// TwinCAT 3 PLC project TcAbbLinkinPLC
// Title: TcAbbLinkin
// Company: Loupe
// Author: Loupe
// ProjectVersion: 0.1.0
// ProgramVersion: 3.1.4024.0
// libraries:
//   Tc2_Standard, * (Beckhoff Automation GmbH)
//   Tc2_System, * (Beckhoff Automation GmbH)
//   Tc2_Utilities, * (Beckhoff Automation GmbH)
//   Tc3_IotBase, * (Beckhoff Automation GmbH)
//   Tc3_JsonXml, * (Beckhoff Automation GmbH)
//   Tc3_Module, * (Beckhoff Automation GmbH)
// project tree:
//   DUTs/ AbbLinkinAuthDigest_Typ.TcDUT, AbbLinkinConfiguration_Typ.TcDUT, AbbLinkinRequestResults_Typ.TcDUT, AbbLinkinRequest_Typ.TcDUT, AbbLinkinRequestQueue_Typ.TcDUT, AbbLinkinRequestStatus_Typ.TcDUT, AbbLinkinAuth_Typ.TcDUT, ABBLINKIN_AUTH_HEADER_VALUE.TcDUT, ABBLINKIN_RWS_API_VERSION.TcDUT, ABBLINKIN_STATE.TcDUT, ABBLINKIN_COMMAND_TYPE.TcDUT, ABBLINKIN_DATA_TYPE_Typ.TcDUT, ABBLINKIN_STRING_EX_LEN.TcDUT (not stored)
//   / PlcTask.TcTTO
//   POUs/ MAIN.TcPOU, Example.TcPOU, TcAbbLinkin.TcPOU
// real-time tasks:
//   TASK PlcTask: cycle T#10ms, priority 20, ADS port 350

CONFIGURATION TcAbbLinkinPLC
    RESOURCE PLC ON TwinCAT3
        TASK PlcTask(INTERVAL := T#10ms, PRIORITY := 20);
        PROGRAM MAIN WITH PlcTask : MAIN;
    END_RESOURCE
END_CONFIGURATION

// ---- DUTs/AbbLinkinAuthDigest_Typ.TcDUT
// Copyright (c) 2024 Loupe (https://loupe.team), provided under the MIT License.
TYPE AbbLinkinAuthDigest_Typ :
STRUCT
	realm : STRING;
	qop : STRING;
	nonce : STRING;
	opaque : STRING;
	nc : STRING;
	cnonce : STRING;
	response : STRING;
	authContent : ABBLINKIN_STRING_EX_LEN;
END_STRUCT
END_TYPE

// ---- DUTs/AbbLinkinConfiguration_Typ.TcDUT
// Copyright (c) 2024 Loupe (https://loupe.team), provided under the MIT License.
TYPE AbbLinkinConfiguration_Typ :
STRUCT
	rwsIpAddress : STRING := '127.0.0.1';
	rwsTcpPort : USINT := 80;
	rwsVersion : ABBLINKIN_RWS_API_VERSION;
	rwsUsername : STRING := 'Default User';
	rwsPassword : STRING := 'robotics';
	tlsAllowRwsCertSelfSigned : BOOL := FALSE;
	tlsCAFile : STRING := '';
END_STRUCT
END_TYPE

// ---- DUTs/AbbLinkinRequestResults_Typ.TcDUT
// Copyright (c) 2024 Loupe (https://loupe.team), provided under the MIT License.
TYPE AbbLinkinRequestResults_Typ :
STRUCT
	pDataBool	: POINTER TO BOOL;
	pDataDint	: POINTER TO DINT;
	pDataLreal	: POINTER TO LREAL;
	pDataString	: POINTER TO STRING;
	dataType	: ABBLINKIN_DATA_TYPE_Typ;
	dataLen		: INT;
END_STRUCT
END_TYPE

// ---- DUTs/AbbLinkinRequest_Typ.TcDUT
// Copyright (c) 2024 Loupe (https://loupe.team), provided under the MIT License.
TYPE AbbLinkinRequest_Typ :
STRUCT
	command : ABBLINKIN_COMMAND_TYPE;
	uri : STRING;
	httpMethod : ETcIotHttpRequestType;
	httpBody : ABBLINKIN_STRING_EX_LEN := '';
	pStatus : POINTER TO AbbLinkinRequestStatus_Typ;
	results : AbbLinkinRequestResults_Typ;
END_STRUCT
END_TYPE

// ---- DUTs/AbbLinkinRequestQueue_Typ.TcDUT
// Copyright (c) 2024 Loupe (https://loupe.team), provided under the MIT License.
TYPE AbbLinkinRequestQueue_Typ :
STRUCT
	request : AbbLinkinRequest_Typ;
	empty : BOOL := TRUE;
END_STRUCT
END_TYPE

// ---- DUTs/AbbLinkinRequestStatus_Typ.TcDUT
// Copyright (c) 2024 Loupe (https://loupe.team), provided under the MIT License.
TYPE AbbLinkinRequestStatus_Typ :
STRUCT
	busy		: BOOL;
	done		: BOOL;
	error		: BOOL;
	errorID		: DINT;
	errorMsg	: STRING;
END_STRUCT
END_TYPE

// ---- DUTs/AbbLinkinAuth_Typ.TcDUT
// Copyright (c) 2024 Loupe (https://loupe.team), provided under the MIT License.
TYPE AbbLinkinAuth_Typ :
STRUCT
	numAttempts : UINT;
	wwwAuthContent : ABBLINKIN_STRING_EX_LEN;
	digest : AbbLinkinAuthDigest_Typ;
	httpSessionCookie : STRING;
	ABBCXCookie : STRING;
END_STRUCT
END_TYPE

// ---- DUTs/ABBLINKIN_AUTH_HEADER_VALUE.TcDUT
{attribute 'qualified_only'}
{attribute 'strict'}
TYPE ABBLINKIN_AUTH_HEADER_VALUE :
(
	NONE,
	BASIC,
	DIGEST
);
END_TYPE

// ---- DUTs/ABBLINKIN_RWS_API_VERSION.TcDUT
{attribute 'qualified_only'}
{attribute 'strict'}
TYPE ABBLINKIN_RWS_API_VERSION :
(
	V1 := 0,
	V2 := 2
);
END_TYPE

// ---- DUTs/ABBLINKIN_STATE.TcDUT
// Copyright (c) 2024 Loupe (https://loupe.team), provided under the MIT License.
{attribute 'qualified_only'}
{attribute 'strict'}
TYPE ABBLINKIN_STATE :
(
	IDLE,
	SEND_REQUEST,
	WAIT_FOR_RESONSE,
	PROCESS_RESPONSE,
	AUTH_START,
	AUTH_SEND_REQUEST,
	AUTH_WAIT_FOR_RESONSE,
	AUTH_PROCESS_RESPONSE,
	AUTH_DIGEST_RESPONSE_CALCULATE,
	AUTH_DIGEST_RESPONSE_SEND
);
END_TYPE

// ---- DUTs/ABBLINKIN_COMMAND_TYPE.TcDUT
// Copyright (c) 2024 Loupe (https://loupe.team), provided under the MIT License.
{attribute 'qualified_only'}
{attribute 'strict'}
TYPE ABBLINKIN_COMMAND_TYPE :
(
	GET_IO,
	GET_PANEL_CTRL_STATE,
	GET_PANEL_OP_MODE,
	GET_RAPID_STATE,
	GET_SYMBOL,
	POWER_OFF,
	POWER_ON,
	RAPID_RESET,
	RAPID_START,
	RAPID_STOP,
	SET_IO,
	SET_SYMBOL
);
END_TYPE

// ---- DUTs/ABBLINKIN_DATA_TYPE_Typ.TcDUT
// Copyright (c) 2024 Loupe (https://loupe.team), provided under the MIT License.
{attribute 'qualified_only'}
{attribute 'strict'}
TYPE ABBLINKIN_DATA_TYPE_Typ :
(
	_NONE,
	_STRING,
	_BOOL,
	_DINT,
	_LREAL
);
END_TYPE

// ---- POUs/MAIN.TcPOU
// Copyright (c) 2024 Loupe (https://loupe.team), provided under the MIT License.
PROGRAM MAIN
VAR
	myRobotLink : TcAbbLinkin;
	userSetConfigurationNow : BOOL := TRUE;
	userConnectStartNow : BOOL := TRUE;
	userConnectStopNow : BOOL;
	
	userGetPanelCtrlStateNow : BOOL;
	userGetPanelCtrlStateStatus : AbbLinkinRequestStatus_Typ;
	userGetPanelCtrlStateResult : STRING;
	
	userGetPanelOpModeNow : BOOL;
	userGetPanelOpModeStatus : AbbLinkinRequestStatus_Typ;
	userGetPanelOpModeResult : STRING;
	
	userGetRapidStateNow : BOOL;
	userGetRapidStateStatus : AbbLinkinRequestStatus_Typ;
	userGetRapidStateResult : STRING;
	
	userGetIoBoolNow : BOOL;
	userGetIoBoolStatus : AbbLinkinRequestStatus_Typ;
	userGetIoBoolResult : BOOL;
	
	userGetIoLrealNow : BOOL;
	userGetIoLrealStatus : AbbLinkinRequestStatus_Typ;
	userGetIoLrealResult : LREAL;
	
	userGetIoDintNow : BOOL;
	userGetIoDintStatus : AbbLinkinRequestStatus_Typ;
	userGetIoDintResult : DINT;
	
	
	userSetIoBoolNow : BOOL;
	userSetIoBoolValue : BOOL := 1;
	userSetIoBoolStatus : AbbLinkinRequestStatus_Typ;
	userSetIoDintNow : BOOL;
	userSetIoDintValue : DINT := 57;
	userSetIoDintStatus : AbbLinkinRequestStatus_Typ;
	userSetIoLrealNow : BOOL;
	userSetIoLrealValue : LREAL := 41.123456;
	userSetIoLrealStatus : AbbLinkinRequestStatus_Typ;
	
	
	userGetSymbolBoolNow : BOOL;
	userGetSymbolBoolResult : BOOL;
	userGetSymbolBoolStatus : AbbLinkinRequestStatus_Typ;
	userGetSymbolNumNow : BOOL;
	userGetSymbolNumResult : LREAL;
	userGetSymbolNumStatus : AbbLinkinRequestStatus_Typ;
	userGetSymbolStringNow : BOOL;
	userGetSymbolStringResult : STRING;
	userGetSymbolStringStatus : AbbLinkinRequestStatus_Typ;
	
	userSetSymbolBoolNow : BOOL;
	userSetSymbolBoolValue : BOOL := 1;
	userSetSymbolBoolStatus : AbbLinkinRequestStatus_Typ;
	userSetSymbolDintNow : BOOL;
	userSetSymbolDintValue : DINT := -57;
	userSetSymbolDintStatus : AbbLinkinRequestStatus_Typ;
	userSetSymbolLrealNow : BOOL;
	userSetSymbolLrealValue : LREAL := -41.123456;
	userSetSymbolLrealStatus : AbbLinkinRequestStatus_Typ;
	userSetSymbolStringNow : BOOL;
	userSetSymbolStringValue : STRING := 'test String';
	userSetSymbolStringStatus : AbbLinkinRequestStatus_Typ;
	userSetSymbolWStringNow : BOOL;
	userSetSymbolWStringValue : WSTRING := "test WString";
	userSetSymbolWStringStatus : AbbLinkinRequestStatus_Typ;
	
	
	userPowerOffNow : BOOL;
	userPowerOffStatus : AbbLinkinRequestStatus_Typ;
	userPowerOnNow : BOOL;
	userPowerOnStatus : AbbLinkinRequestStatus_Typ;
	userRapidResetNow : BOOL;
	userRapidResetStatus : AbbLinkinRequestStatus_Typ;
	userRapidStopNow : BOOL;
	userRapidStopStatus : AbbLinkinRequestStatus_Typ;
	userRapidStartNow : BOOL;
	userRapidStartStatus : AbbLinkinRequestStatus_Typ;
	
	
	userAckErrorNow : BOOL;
END_VAR


// Set configuration
if userSetConfigurationNow then
	myRobotLink.configuration.rwsIpAddress := '127.0.0.1';
	myRobotLink.configuration.rwsTcpPort := 80;
	myRobotLink.configuration.rwsVersion := ABBLINKIN_RWS_API_VERSION.V2;
	myRobotLink.configuration.rwsUsername := 'Default User';
	myRobotLink.configuration.rwsPassword := 'robotics';
	//myRobotLink.configuration.tlsAllowRwsCertSelfSigned := TRUE;
	myRobotLink.configuration.tlsAllowRwsCertSelfSigned := FALSE;
	myRobotLink.configuration.tlsCAFile := 'C:\TwinCAT\3.1\Config\Certificates\TcAbbLinkinCA.pem';
	
	userSetConfigurationNow := FALSE;
END_IF


// Cyclic
myRobotLink.Cyclic();


IF userConnectStartNow THEN
	myRobotLink.Connect();
	userConnectStartNow := FALSE;
END_IF

IF userConnectStopNow THEN
	myRobotLink.Disconnect();
	userConnectStopNow := FALSE;
END_IF


IF userGetPanelCtrlStateNow THEN
	myRobotLink.GetPanelCtrlState(ADR(userGetPanelCtrlStateStatus), ADR(userGetPanelCtrlStateResult));
	userGetPanelCtrlStateNow := FALSE;
END_IF


IF userGetPanelOpModeNow THEN
	myRobotLink.GetPanelOpMode(ADR(userGetPanelOpModeStatus), ADR(userGetPanelOpModeResult));
	userGetPanelOpModeNow := FALSE;
END_IF


IF userGetRapidStateNow THEN
	myRobotLink.GetRapidState(ADR(userGetRapidStateStatus), ADR(userGetRapidStateResult));
	userGetRapidStateNow := FALSE;
END_IF


IF userGetIoBoolNow THEN
	myRobotLink.GetIODigital(signal := 'myInputDIG', pStatus := ADR(userGetIoBoolStatus), pResult := ADR(userGetIoBoolResult));
	userGetIoBoolNow := FALSE;
END_IF

IF userGetIoLrealNow THEN
	myRobotLink.GetIOAnalog(signal := 'myInputANA', pStatus := ADR(userGetIoLrealStatus), pResult := ADR(userGetIoLrealResult));
	userGetIoLrealNow := FALSE;
END_IF

IF userGetIoDintNow THEN
	myRobotLink.GetIOGroup(signal := 'myInputGRP', pStatus := ADR(userGetIoDintStatus), pResult := ADR(userGetIoDintResult));
	userGetIoDintNow := FALSE;
END_IF


IF userSetIoBoolNow THEN
	myRobotLink.SetIO('myInputDIG', userSetIoBoolValue, ADR(userSetIoBoolStatus));
	userSetIoBoolNow := FALSE;
END_IF
IF userSetIoDintNow THEN
	myRobotLink.SetIO('myInputGRP', userSetIoDintValue, ADR(userSetIoDintStatus));
	userSetIoDintNow := FALSE;
END_IF
IF userSetIoLrealNow THEN
	myRobotLink.SetIO('myInputANA', userSetIoLrealValue, ADR(userSetIoLrealStatus));
	userSetIoLrealNow := FALSE;
END_IF


IF userGetSymbolBoolNow THEN
	myRobotLink.GetSymbolBool(symbolUrl := 'RAPID/T_ROB1/Module1/myRapidBool', pStatus := ADR(userGetSymbolBoolStatus), pResult := ADR(userGetSymbolBoolResult));
	userGetSymbolBoolNow := FALSE;
END_IF
IF userGetSymbolNumNow THEN
	myRobotLink.GetSymbolNum(symbolUrl := 'RAPID/T_ROB1/Module1/myRapidNum', pStatus := ADR(userGetSymbolNumStatus), pResult := ADR(userGetSymbolNumResult));
	userGetSymbolNumNow := FALSE;
END_IF
IF userGetSymbolStringNow THEN
	myRobotLink.GetSymbolString(symbolUrl := 'RAPID/T_ROB1/Module1/myRapidString', pStatus := ADR(userGetSymbolStringStatus), pResult := ADR(userGetSymbolStringResult));
	userGetSymbolStringNow := FALSE;
END_IF


IF userSetSymbolBoolNow THEN
	myRobotLink.SetSymbol('RAPID/T_ROB1/Module1/myRapidBool', userSetSymbolBoolValue, ADR(userSetSymbolBoolStatus));
	userSetSymbolBoolNow := FALSE;
END_IF
IF userSetSymbolDintNow THEN
	myRobotLink.SetSymbol('RAPID/T_ROB1/Module1/myRapidNum', userSetSymbolDintValue, ADR(userSetSymbolDintStatus));
	userSetSymbolDintNow := FALSE;
END_IF
IF userSetSymbolLrealNow THEN
	myRobotLink.SetSymbol('RAPID/T_ROB1/Module1/myRapidNum', userSetSymbolLrealValue, ADR(userSetSymbolLrealStatus));
	userSetSymbolLrealNow := FALSE;
END_IF
IF userSetSymbolStringNow THEN
	myRobotLink.SetSymbol('RAPID/T_ROB1/Module1/myRapidString', userSetSymbolStringValue, ADR(userSetSymbolStringStatus));
	userSetSymbolStringNow := FALSE;
END_IF
IF userSetSymbolWStringNow THEN
	myRobotLink.SetSymbol('RAPID/T_ROB1/Module1/myRapidString', userSetSymbolWStringValue, ADR(userSetSymbolWStringStatus));
	userSetSymbolWStringNow := FALSE;
END_IF


IF userPowerOffNow THEN
	myRobotLink.PowerOff(ADR(userPowerOffStatus));
	userPowerOffNow := FALSE;
END_IF
IF userPowerOnNow THEN
	myRobotLink.PowerOn(ADR(userPowerOnStatus));
	userPowerOnNow := FALSE;
END_IF
IF userRapidResetNow THEN
	myRobotLink.RapidReset(ADR(userRapidResetStatus));
	userRapidResetNow := FALSE;
END_IF
IF userRapidStopNow THEN
	myRobotLink.RapidStop(ADR(userRapidStopStatus));
	userRapidStopNow := FALSE;
END_IF
IF userRapidStartNow THEN
	myRobotLink.RapidStart(ADR(userRapidStartStatus));
	userRapidStartNow := FALSE;
END_IF


IF userAckErrorNow THEN
	myRobotLink.AckError();
	userAckErrorNow := FALSE;
END_IF

END_PROGRAM

// ---- POUs/TcAbbLinkin.TcPOU
// Copyright (c) 2024 Loupe (https://loupe.team), provided under the MIT License.
FUNCTION_BLOCK TcAbbLinkin
VAR_INPUT
	configuration : AbbLinkinConfiguration_Typ;
END_VAR
VAR_OUTPUT
	readyForCmd : BOOL;
	error : BOOL;
	errorID : DINT;
	errorMsg : STRING;
END_VAR
VAR
	_connectionEnable : BOOL;
	_sendingEnabled : BOOL;
	_authorized : BOOL;
	
	_httpClient : FB_IotHttpClient;
	_httpRequest : FB_IotHttpRequest;
	_httpHeader : FB_IotHttpHeaderFieldMap;
	
	_methodConnectionStartCalled : BOOL;
	_methodConnectionStopCalled : BOOL;
	_methodAckErrorCalled : BOOL;
	
	_state : ABBLINKIN_STATE;
	_auth : AbbLinkinAuth_Typ;
	_requestQueue : AbbLinkinRequestQueue_Typ;
	_currentRequest : AbbLinkinRequest_Typ;
	_numRequestAttempts : UINT;
END_VAR

VAR CONSTANT
	AUTH_URI : STRING := '/?json=1';
	MAX_REQUESTS_ATTEMPTS : UINT := 3;
END_VAR

// Copyright (c) 2024 Loupe (https://loupe.team), provided under the MIT License.
METHOD PRIVATE _calculateDigestResponse : STRING
VAR_INPUT
	username : STRING;
	realm : STRING;
	password : STRING;
	httpMethod : STRING;
	uri : STRING;
	nonce : STRING;
	nc : STRING;
	cnonce : STRING;
	qop : STRING;
END_VAR

VAR
	tempString : ABBLINKIN_STRING_EX_LEN;
	h1_byArr : ARRAY[0..15] OF BYTE;
	h1_hexStr : STRING;
	h2_byArr : ARRAY[0..15] OF BYTE;
	h2_hexStr : STRING;
	response_byArr : ARRAY[0..15] OF BYTE;
	response_hexStr : STRING;
	i : INT;
END_VAR

// H1 hash
tempString := '';
tempString := CONCAT(tempString, username);
tempString := CONCAT(tempString, ':');
tempString := CONCAT(tempString, realm);
tempString := CONCAT(tempString, ':');
tempString := CONCAT(tempString, password);
F_GenerateHashValue(E_HashMode.HASH_MD5, ADR(tempString), INT_TO_UDINT(LEN(tempString)), ADR(h1_byArr), SIZEOF(h1_byArr));
h1_hexStr := '';
FOR i := 0 TO 15 DO
	h1_hexStr := CONCAT(h1_hexStr, BYTE_TO_HEXSTR(h1_byArr[i], 2, TRUE));
END_FOR


// H2 Hash
tempString := '';
tempString := CONCAT(tempString, httpMethod);
tempString := CONCAT(tempString, ':');
tempString := CONCAT(tempString, uri);
F_GenerateHashValue(E_HashMode.HASH_MD5, ADR(tempString), INT_TO_UDINT(LEN(tempString)), ADR(h2_byArr), SIZEOF(h2_byArr));
h2_hexStr := '';
FOR i := 0 TO 15 DO
	h2_hexStr := CONCAT(h2_hexStr, BYTE_TO_HEXSTR(h2_byArr[i], 2, TRUE));
END_FOR


// Response hash
tempString := '';
tempString := CONCAT(tempString, h1_hexStr);
tempString := CONCAT(tempString, ':');
tempString := CONCAT(tempString, nonce);
tempString := CONCAT(tempString, ':');
tempString := CONCAT(tempString, nc);
tempString := CONCAT(tempString, ':');
tempString := CONCAT(tempString, cnonce);
tempString := CONCAT(tempString, ':');
tempString := CONCAT(tempString, qop);
tempString := CONCAT(tempString, ':');
tempString := CONCAT(tempString, h2_hexStr);
F_GenerateHashValue(E_HashMode.HASH_MD5, ADR(tempString), INT_TO_UDINT(LEN(tempString)), ADR(response_byArr), SIZEOF(response_byArr));
response_hexStr := '';
FOR i := 0 TO 15 DO
	response_hexStr := CONCAT(response_hexStr, BYTE_TO_HEXSTR(response_byArr[i], 2, TRUE));
END_FOR

_calculateDigestResponse := response_hexStr;
END_METHOD

// Copyright (c) 2024 Loupe (https://loupe.team), provided under the MIT License.
METHOD PRIVATE _callCommandSuccessHandler : BOOL
VAR_IN_OUT
	request : AbbLinkinRequest_Typ;
	httpRequest : FB_IotHttpRequest;
END_VAR

CASE request.command OF 
	ABBLINKIN_COMMAND_TYPE.GET_IO:
		_getIORespCallbackSuccess(httpRequest, request);
		
	ABBLINKIN_COMMAND_TYPE.GET_CTRL_STATE:
		_getCtrlStateRespCallbackSuccess(httpRequest, request);
		
	ABBLINKIN_COMMAND_TYPE.GET_OP_MODE:
		_getOpModeRespCallbackSuccess(httpRequest, request);
		
	ABBLINKIN_COMMAND_TYPE.GET_RAPID_STATE:
		_getRapidStateRespCallbackSuccess(httpRequest, request);
		
	ABBLINKIN_COMMAND_TYPE.GET_SYMBOL:
		_getSymbolRespCallbackSuccess(httpRequest, request);
		
	ABBLINKIN_COMMAND_TYPE.POWER_OFF:
		;// Do Nothing
		
	ABBLINKIN_COMMAND_TYPE.POWER_ON:
		;// Do Nothing
		
	ABBLINKIN_COMMAND_TYPE.RAPID_RESET:
		;// Do Nothing
		
	ABBLINKIN_COMMAND_TYPE.RAPID_START:
		;// Do Nothing
		
	ABBLINKIN_COMMAND_TYPE.RAPID_STOP:
		;// Do Nothing
		
	ABBLINKIN_COMMAND_TYPE.SET_IO:
		;// Do Nothing
		
	ABBLINKIN_COMMAND_TYPE.SET_SYMBOL:
		;// Do Nothing
		
END_CASE
END_METHOD

// Copyright (c) 2024 Loupe (https://loupe.team), provided under the MIT License.
METHOD PRIVATE _clearRequestStatus : BOOL
VAR_INPUT
	pStatus : POINTER TO AbbLinkinRequestStatus_Typ;
END_VAR

pStatus^.busy := FALSE;
pStatus^.done := FALSE;
pStatus^.error := FALSE;
pStatus^.errorID := 0;
pStatus^.errorMsg := '';

_clearRequestStatus := TRUE;
END_METHOD

// Copyright (c) 2024 Loupe (https://loupe.team), provided under the MIT License.
METHOD PRIVATE _configureClient : BOOL
VAR_IN_OUT
	connectionConfig : AbbLinkinConfiguration_Typ;	
END_VAR

_httpClient.sHostName := connectionConfig.rwsIpAddress;
_httpClient.nHostPort := connectionConfig.rwsTcpPort;
_httpClient.bKeepAlive := TRUE;
_httpClient.tConnectionTimeout := T#10S;


CASE connectionConfig.rwsVersion OF
	ABBLINKIN_RWS_API_VERSION.V1:
		_httpClient.stTLS.bNoServerCertCheck := FALSE;
		
	ABBLINKIN_RWS_API_VERSION.V2:
		IF connectionConfig.tlsAllowRwsCertSelfSigned THEN 
			_httpClient.stTLS.bNoServerCertCheck := TRUE;
		ELSE
			_httpClient.stTLS.bNoServerCertCheck := FALSE;
			_httpClient.stTLS.sCA := connectionConfig.tlsCAFile;
		END_IF
END_CASE
END_METHOD

// Copyright (c) 2024 Loupe (https://loupe.team), provided under the MIT License.
METHOD PRIVATE _encodeBase64 : STRING
VAR_INPUT
	rawText : STRING;
END_VAR
VAR
	_jsonDomParser : FB_JsonDomParser;
	_jsonRoot : SJsonValue;
	_jsonValue : SJsonValue;
	_jsonValue2 : SJsonValue;
END_VAR
	
_jsonRoot := _jsonDomParser.ParseDocument('{"k": ""}');
_jsonValue := _jsonDomParser.FindMember(_jsonRoot, 'k');
_jsonValue2 := _jsonDomParser.SetBase64(_jsonValue, ADR(rawText), LEN(rawText));
_encodeBase64 := _jsonDomParser.GetString(_jsonValue2);
END_METHOD

METHOD PRIVATE _generateCnonce : STRING
VAR_INPUT
END_VAR

_generateCnonce := 'diddLOPR';	// TODO: reimplement with random generation
END_METHOD

// Copyright (c) 2024 Loupe (https://loupe.team), provided under the MIT License.
METHOD PRIVATE _getCtrlStateRespCallbackSuccess : BOOL
VAR_IN_OUT
	httpRequest : FB_IotHttpRequest;
	request : AbbLinkinRequest_Typ;
END_VAR
VAR
	jsonDomParser : FB_JsonDomParser;
	jsonRoot : SJsonValue;
	jsonValue : SJsonValue;
	valuePath : STRING;
	tempString : STRING;
END_VAR
CASE configuration.rwsVersion OF 
	ABBLINKIN_RWS_API_VERSION.V1:
		valuePath := '_embedded/_state#0/ctrlstate';
	ABBLINKIN_RWS_API_VERSION.V2:
		valuePath := 'state#0/ctrlstate';
END_CASE

jsonRoot := httpRequest.GetJsonDomContent(jsonDomParser);
jsonValue := jsonDomParser.FindMemberPath(jsonRoot, valuePath);
IF (jsonValue <> 0) THEN
	request.results.pDataString^ := jsonDomParser.GetString(jsonValue);
ELSE
	request.pStatus^.error := TRUE;
	request.pStatus^.errorID := 0;
	request.pStatus^.errorMsg := 'Unable to parse RWS json response';
END_IF


_getCtrlStateRespCallbackSuccess := TRUE;
END_METHOD

// Copyright (c) 2024 Loupe (https://loupe.team), provided under the MIT License.
METHOD PRIVATE _getIO : BOOL
VAR_INPUT
	signal : STRING;
	pStatus : POINTER TO AbbLinkinRequestStatus_Typ;
	pResultBool : POINTER TO BOOL := 0;
	pResultDint : POINTER TO DINT := 0;
	pResultLreal : POINTER TO LREAL := 0;
END_VAR

VAR
	request : AbbLinkinRequest_Typ;
	pointersSet : INT;
END_VAR

VAR CONSTANT
	THIS_COMMAND_TYPE: ABBLINKIN_COMMAND_TYPE := ABBLINKIN_COMMAND_TYPE.GET_IO;
END_VAR
IF pStatus = 0 THEN
	_getIO := FALSE;
	RETURN;
END_IF

// Clear Status
_clearRequestStatus(pStatus);

// Check that one and only one pointer is populated
pointersSet := 0;
IF (pResultBOOL <> 0) THEN 
	request.results.dataType := ABBLINKIN_DATA_TYPE_Typ._BOOL;
	request.results.pDataBool := pResultBool;
	pointersSet := pointersSet + 1; 
END_IF
IF (pResultDINT <> 0) THEN
	request.results.dataType := ABBLINKIN_DATA_TYPE_Typ._DINT;
	request.results.pDataDint := pResultDint;
	pointersSet := pointersSet + 1;
END_IF
IF (pResultLREAL <> 0) THEN
	request.results.dataType := ABBLINKIN_DATA_TYPE_Typ._LREAL;
	request.results.pDataLreal := pResultLreal;
	pointersSet := pointersSet + 1;
END_IF


IF pointersSet = 0 THEN
	pStatus^.error := TRUE;
	pStatus^.errorMsg := TO_STRING(THIS_COMMAND_TYPE);
	pStatus^.errorMsg := CONCAT(pStatus^.errorMsg, ' : No result pointer set');
	_getIO := FALSE;
ELSIF pointersSet >= 2 THEN
	pStatus^.error := TRUE;
	pStatus^.errorMsg := TO_STRING(THIS_COMMAND_TYPE);
	pStatus^.errorMsg := CONCAT(pStatus^.errorMsg, ' : Two or more result pointer set');
	_getIO := FALSE;
END_IF

request.pStatus := pStatus;
request.command := THIS_COMMAND_TYPE;
request.httpMethod :=  ETcIotHttpRequestType.HTTP_Get;

CASE configuration.rwsVersion OF
	ABBLINKIN_RWS_API_VERSION.V1:
		request.uri := '/rw/iosystem/signals/';
		request.uri := CONCAT(request.uri, signal);
		request.uri := CONCAT(request.uri, '?json=1');

	ABBLINKIN_RWS_API_VERSION.V2:	
		request.uri := '/rw/iosystem/signals/';
		request.uri := CONCAT(request.uri, signal);
END_CASE

// Add Request to Queue, and Set Busy (or Error) Status
IF _requestQueueAdd(request) THEN
	pStatus^.busy := TRUE;
	_getIO := TRUE;
ELSE
	pStatus^.error := TRUE;
	pStatus^.errorMsg := TO_STRING(THIS_COMMAND_TYPE);
	pStatus^.errorMsg := CONCAT(pStatus^.errorMsg, ' could not be added to request Queue');
	_getIO := FALSE;
END_IF
END_METHOD

// Copyright (c) 2024 Loupe (https://loupe.team), provided under the MIT License.
METHOD PRIVATE _getIORespCallbackSuccess : BOOL
VAR_IN_OUT
	httpRequest : FB_IotHttpRequest;
	request : AbbLinkinRequest_Typ;
END_VAR
VAR
	jsonDomParser : FB_JsonDomParser;
	jsonRoot : SJsonValue;
	jsonValue : SJsonValue;
	valuePath : STRING;
	valueString : STRING;
END_VAR

CASE configuration.rwsVersion OF 
	ABBLINKIN_RWS_API_VERSION.V1:
		valuePath := '_embedded/_state#0/lvalue';
	ABBLINKIN_RWS_API_VERSION.V2:
		valuePath := '_embedded/resources#0/lvalue';
END_CASE

jsonRoot := httpRequest.GetJsonDomContent(jsonDomParser);
jsonValue := jsonDomParser.FindMemberPath(jsonRoot, valuePath);
IF (jsonValue <> 0) THEN
	valueString := jsonDomParser.GetString(jsonValue);
	
	CASE request.results.dataType OF
		ABBLINKIN_DATA_TYPE_Typ._BOOL:
			request.results.pDataBool^ := INT_TO_BOOL(STRING_TO_INT(valueString));
		ABBLINKIN_DATA_TYPE_Typ._DINT:
			request.results.pDataDint^ := STRING_TO_DINT(valueString);
		ABBLINKIN_DATA_TYPE_Typ._LREAL:
			request.results.pDataLreal^ := STRING_TO_LREAL(valueString);
	END_CASE
ELSE
	request.pStatus^.error := TRUE;
	request.pStatus^.errorID := 0;
	request.pStatus^.errorMsg := 'Unable to parse RWS json response';
END_IF


_getIORespCallbackSuccess := TRUE;
END_METHOD

// Copyright (c) 2024 Loupe (https://loupe.team), provided under the MIT License.
METHOD PRIVATE _getOpModeRespCallbackSuccess : BOOL
VAR_IN_OUT
	httpRequest : FB_IotHttpRequest;
	request : AbbLinkinRequest_Typ;
END_VAR
VAR
	jsonDomParser : FB_JsonDomParser;
	jsonRoot : SJsonValue;
	jsonValue : SJsonValue;
	valuePath : STRING;
	tempString : STRING;
END_VAR
CASE configuration.rwsVersion OF 
	ABBLINKIN_RWS_API_VERSION.V1:
		valuePath := '_embedded/_state#0/opmode';
	ABBLINKIN_RWS_API_VERSION.V2:
		valuePath := 'state#0/opmode';
END_CASE

jsonRoot := httpRequest.GetJsonDomContent(jsonDomParser);
jsonValue := jsonDomParser.FindMemberPath(jsonRoot, valuePath);
IF (jsonValue <> 0) THEN
	request.results.pDataString^ := jsonDomParser.GetString(jsonValue);
ELSE
	request.pStatus^.error := TRUE;
	request.pStatus^.errorID := 0;
	request.pStatus^.errorMsg := 'Unable to parse RWS json response';
END_IF


_getOpModeRespCallbackSuccess := TRUE;
END_METHOD

// Copyright (c) 2024 Loupe (https://loupe.team), provided under the MIT License.
METHOD PRIVATE _getRapidStateRespCallbackSuccess : BOOL
VAR_IN_OUT
	httpRequest : FB_IotHttpRequest;
	request : AbbLinkinRequest_Typ;
END_VAR
VAR
	jsonDomParser : FB_JsonDomParser;
	jsonRoot : SJsonValue;
	jsonValue : SJsonValue;
	valuePath : STRING;
	tempString : STRING;
END_VAR
CASE configuration.rwsVersion OF 
	ABBLINKIN_RWS_API_VERSION.V1:
		valuePath := '_embedded/_state#0/ctrlexecstate';
	ABBLINKIN_RWS_API_VERSION.V2:
		valuePath := 'state#0/ctrlexecstate';
END_CASE

jsonRoot := httpRequest.GetJsonDomContent(jsonDomParser);
jsonValue := jsonDomParser.FindMemberPath(jsonRoot, valuePath);
IF (jsonValue <> 0) THEN
	request.results.pDataString^ := jsonDomParser.GetString(jsonValue);
ELSE
	request.pStatus^.error := TRUE;
	request.pStatus^.errorID := 0;
	request.pStatus^.errorMsg := 'Unable to parse RWS json response';
END_IF


_getRapidStateRespCallbackSuccess := TRUE;
END_METHOD

// Copyright (c) 2024 Loupe (https://loupe.team), provided under the MIT License.
METHOD PRIVATE _getSymbol : BOOL
VAR_INPUT
	symbolUrl : STRING;
	pStatus : POINTER TO AbbLinkinRequestStatus_Typ;
	pResultBool : POINTER TO BOOL := 0;
	pResultLreal : POINTER TO LREAL := 0;
	pResultString : POINTER TO STRING := 0;
END_VAR

VAR
	request : AbbLinkinRequest_Typ;
	pointersSet : INT;
END_VAR

VAR CONSTANT
	THIS_COMMAND_TYPE: ABBLINKIN_COMMAND_TYPE := ABBLINKIN_COMMAND_TYPE.GET_SYMBOL;
END_VAR
IF pStatus = 0 THEN
	_getSymbol := FALSE;
	RETURN;
END_IF

// Clear Status
_clearRequestStatus(pStatus);

// Check that one and only one pointer is populated
pointersSet := 0;
IF (pResultBOOL <> 0) THEN 
	request.results.dataType := ABBLINKIN_DATA_TYPE_Typ._BOOL;
	request.results.pDataBool := pResultBool;
	pointersSet := pointersSet + 1; 
END_IF
IF (pResultLREAL <> 0) THEN
	request.results.dataType := ABBLINKIN_DATA_TYPE_Typ._LREAL;
	request.results.pDataLreal := pResultLreal;
	pointersSet := pointersSet + 1;
END_IF
IF (pResultSTRING <> 0) THEN
	request.results.dataType := ABBLINKIN_DATA_TYPE_Typ._STRING;
	request.results.pDataString := pResultString;
	pointersSet := pointersSet + 1;
END_IF


IF pointersSet = 0 THEN
	pStatus^.error := TRUE;
	pStatus^.errorMsg := TO_STRING(THIS_COMMAND_TYPE);
	pStatus^.errorMsg := CONCAT(pStatus^.errorMsg, ' : No result pointer set');
	_getSymbol := FALSE;
ELSIF pointersSet >= 2 THEN
	pStatus^.error := TRUE;
	pStatus^.errorMsg := TO_STRING(THIS_COMMAND_TYPE);
	pStatus^.errorMsg := CONCAT(pStatus^.errorMsg, ' : Two or more result pointer set');
	_getSymbol := FALSE;
END_IF

request.pStatus := pStatus;
request.command := THIS_COMMAND_TYPE;
request.httpMethod :=  ETcIotHttpRequestType.HTTP_Get;

CASE configuration.rwsVersion OF
	ABBLINKIN_RWS_API_VERSION.V1:
		request.uri := '/rw/rapid/symbol/data/';
		request.uri := CONCAT(request.uri, symbolUrl);		// e.g. signal='RAPID/T_ROB1/Module1/myRapidString'
		request.uri := CONCAT(request.uri, '?json=1');

	ABBLINKIN_RWS_API_VERSION.V2:	
		request.uri := '/rw/rapid/symbol/';
		request.uri := CONCAT(request.uri, symbolUrl);		// e.g. signal='RAPID/T_ROB1/Module1/myRapidString'
		request.uri := CONCAT(request.uri, '/data');
		
END_CASE

// Add Request to Queue, and Set Busy (or Error) Status
IF _requestQueueAdd(request) THEN
	pStatus^.busy := TRUE;
	_getSymbol := TRUE;
ELSE
	pStatus^.error := TRUE;
	pStatus^.errorMsg := TO_STRING(THIS_COMMAND_TYPE);
	pStatus^.errorMsg := CONCAT(pStatus^.errorMsg, ' could not be added to request Queue');
	_getSymbol := FALSE;
END_IF
END_METHOD

// Copyright (c) 2024 Loupe (https://loupe.team), provided under the MIT License.
METHOD PRIVATE _getSymbolRespCallbackSuccess : BOOL
VAR_IN_OUT
	httpRequest : FB_IotHttpRequest;
	request : AbbLinkinRequest_Typ;
END_VAR
VAR
	jsonDomParser : FB_JsonDomParser;
	jsonRoot : SJsonValue;
	jsonValue : SJsonValue;
	valuePath : STRING;
	valueString : STRING;
	valueStringNoQuotes : STRING;
END_VAR

CASE configuration.rwsVersion OF 
	ABBLINKIN_RWS_API_VERSION.V1:
		valuePath := '_embedded/_state#0/value';
	ABBLINKIN_RWS_API_VERSION.V2:
		valuePath := 'state#0/value';
END_CASE

jsonRoot := httpRequest.GetJsonDomContent(jsonDomParser);
jsonValue := jsonDomParser.FindMemberPath(jsonRoot, valuePath);
IF (jsonValue <> 0) THEN
	valueString := jsonDomParser.GetString(jsonValue);
	
	CASE request.results.dataType OF
		ABBLINKIN_DATA_TYPE_Typ._BOOL:
			request.results.pDataBool^ := STRING_TO_BOOL(valueString);
		ABBLINKIN_DATA_TYPE_Typ._LREAL:
			request.results.pDataLreal^ := STRING_TO_LREAL(valueString);
		ABBLINKIN_DATA_TYPE_Typ._STRING:
			valueStringNoQuotes := MID(valueString, len(valueString) - 2, 2); // MID removes beginning and ending double-quote (") characters
			request.results.pDataString^ := valueStringNoQuotes;
	END_CASE
ELSE
	request.pStatus^.error := TRUE;
	request.pStatus^.errorID := 0;
	request.pStatus^.errorMsg := 'Unable to parse RWS json response';
END_IF


_getSymbolRespCallbackSuccess := TRUE;
END_METHOD

// Copyright (c) 2024 Loupe (https://loupe.team), provided under the MIT License.
METHOD PRIVATE _parseWwwAuthForParameter : STRING

VAR_INPUT
	keyString : STRING;
END_VAR

VAR_IN_OUT
	contentString : ABBLINKIN_STRING_EX_LEN;
END_VAR

VAR
	contentLen : INT;
	keyLocation : INT;
	firstQuoteLocation : INT;
	secondQuoteLocation : INT;
	tempString : ABBLINKIN_STRING_EX_LEN;
END_VAR

contentLen := LEN(contentString);
keyLocation := FIND(contentString, keyString);
IF keyLocation = 0 THEN 
	_parseWwwAuthForParameter := '';
	RETURN;
END_IF
tempString := RIGHT(contentString, contentLen - keyLocation);
firstQuoteLocation := FIND(tempString, '"') + keyLocation;
tempString := RIGHT(contentString, contentLen - firstQuoteLocation);
secondQuoteLocation := FIND(tempString, '"') + firstQuoteLocation;
_parseWwwAuthForParameter := MID(contentString, secondQuoteLocation - firstQuoteLocation - 1, firstQuoteLocation + 1);
END_METHOD

// Copyright (c) 2024 Loupe (https://loupe.team), provided under the MIT License.
METHOD PRIVATE _requestQueueAdd : BOOL
VAR_INPUT
	request : AbbLinkinRequest_Typ;
END_VAR

// Note : the requestQueue and this method are temporary implementations. It is not a real queue as shown (it can only hold one request).

IF _requestQueue.empty THEN
	_requestQueue.request := request;
	_requestQueue.empty := FALSE;
	_requestQueueAdd := TRUE;
ELSE
	// Do not overwrite request
	_requestQueueAdd := FALSE;
END_IF
END_METHOD

// Copyright (c) 2024 Loupe (https://loupe.team), provided under the MIT License.
METHOD PRIVATE _requestQueuePop : AbbLinkinRequest_Typ
VAR_INPUT
END_VAR

// Note : the requestQueue and this method are temporary implementations. It is not a real queue as shown.

_requestQueue.empty := TRUE;
_requestQueuePop := _requestQueue.request;
END_METHOD

// Copyright (c) 2024 Loupe (https://loupe.team), provided under the MIT License.
METHOD PRIVATE _setHeaders : BOOL
VAR_INPUT
	authorizationValue : ABBLINKIN_AUTH_HEADER_VALUE;
END_VAR
VAR
	authValue : STRING;
	combinedCredentialsRaw : STRING;
	combinedCredentialsBase64 : STRING;
	anyCookieSetYet : BOOL;
	tempString : STRING;
	cookieValue : ABBLINKIN_STRING_EX_LEN;
END_VAR

// Accept 
IF configuration.rwsVersion = ABBLINKIN_RWS_API_VERSION.V2 THEN
	_httpHeader.AddField('Accept', 'application/hal+json;v=2.0', FALSE);
ELSE
	_httpHeader.AddField('Accept', '*/*', FALSE);
END_IF


// Authorization
CASE authorizationValue OF
	ABBLINKIN_AUTH_HEADER_VALUE.NONE:
		_httpHeader.AddField('Authorization', ' ', FALSE);
	
	ABBLINKIN_AUTH_HEADER_VALUE.BASIC:
		combinedCredentialsRaw := configuration.rwsUsername;
		combinedCredentialsRaw := CONCAT(combinedCredentialsRaw, ':');
		combinedCredentialsRaw := CONCAT(combinedCredentialsRaw, configuration.rwsPassword);
		combinedCredentialsBase64 := _encodeBase64(combinedCredentialsRaw);
		
		authValue := 'Basic ';
		authValue := CONCAT(authValue, combinedCredentialsBase64);
		_httpHeader.AddField('Authorization', authValue, FALSE);
	
	ABBLINKIN_AUTH_HEADER_VALUE.DIGEST:
		_httpHeader.AddField('Authorization', _auth.digest.authContent, FALSE);
		
END_CASE


// Cookie
anyCookieSetYet := FALSE;
cookieValue := '';
IF LEN(_auth.httpSessionCookie) > 0 THEN
	tempString := '';
	tempString := CONCAT(tempString, '-http-session-='); 
	tempString := CONCAT(tempString, _auth.httpSessionCookie); 
	cookieValue := CONCAT(cookieValue, tempString);
	anyCookieSetYet := TRUE;
END_IF

IF LEN(_auth.ABBCXCookie) > 0 THEN
	IF anyCookieSetYet THEN
		tempString := '; ';
	ELSE
		tempString := '';	
	END_IF
	tempString := CONCAT(tempString, 'ABBCX='); 
	tempString := CONCAT(tempString, _auth.ABBCXCookie); 
	cookieValue := CONCAT(cookieValue, tempString);
	anyCookieSetYet := TRUE;
END_IF

_httpHeader.AddField('Cookie', cookieValue, FALSE);


// Content-Type
CASE configuration.rwsVersion OF
	ABBLINKIN_RWS_API_VERSION.V1:
		_httpHeader.AddField('Content-Type', 'application/x-www-form-urlencoded', FALSE);
	ABBLINKIN_RWS_API_VERSION.V2:
		_httpHeader.AddField('Content-Type', 'application/x-www-form-urlencoded;v=2.0', FALSE);	
END_CASE
END_METHOD

// Copyright (c) 2024 Loupe (https://loupe.team), provided under the MIT License.
METHOD PRIVATE _storeCookies : BOOL
VAR_INPUT
	httpRequest : FB_IotHttpRequest;
END_VAR
VAR
	setCookieValue : ABBLINKIN_STRING_EX_LEN;
	Set : INT;
	tempString : ABBLINKIN_STRING_EX_LEN;
	setCookieValueLen : INT;
	keyLoc : INT;
	equalLoc : INT;
	semicolonLoc : INT;
END_VAR

IF httpRequest.GetHeaderField('Set-Cookie', ADR(setCookieValue), SIZEOF(setCookieValue)-1) THEN 
	
	// NOTE : if there are multiple 'Set-Cookie' headers, they will all be contained in one value, separated by a newline
	//		e.g. 'token1=Beckhoff$Ntoken2=IoT' per https://infosys.beckhoff.com/content/1033/tf6760_tc3_iot_https_rest/9335286283.html
	// Real header examples from RWS:
	//		Set-Cookie: -http-session-=1: : http.session: : 241eb766f25fa09a53f749ebbafb9aa9; path=/; domain=127.0.0.1; httponly\r\n
	//		Set-Cookie : ABBCX=12; path=/; domain=127.0.0.1; httponly\r\n
	
	setCookieValueLen := len(setCookieValue);
		
	// -http-session-
	keyLoc := FIND(setCookieValue, '-http-session-');
	tempString := RIGHT(setCookieValue, setCookieValueLen - keyLoc);
	equalLoc := FIND(tempString, '=') + keyLoc;
	tempString := RIGHT(setCookieValue, setCookieValueLen - equalLoc);
	semicolonLoc := FIND(tempString, ';') + equalLoc;
	_auth.httpSessionCookie := MID(setCookieValue, semicolonLoc - equalLoc - 1, equalLoc + 1);
	
	
	// ABBCX
	keyLoc := FIND(setCookieValue, 'ABBCX');
	tempString := RIGHT(setCookieValue, setCookieValueLen - keyLoc);
	equalLoc := FIND(tempString, '=') + keyLoc;
	tempString := RIGHT(setCookieValue, setCookieValueLen - equalLoc);
	semicolonLoc := FIND(tempString, ';') + equalLoc;
	_auth.ABBCXCookie := MID(setCookieValue, semicolonLoc - equalLoc - 1, equalLoc + 1);
	
	
END_IF
END_METHOD

// Copyright (c) 2024 Loupe (https://loupe.team), provided under the MIT License.
METHOD AckError
VAR_INPUT
END_VAR

_methodAckErrorCalled := TRUE;
END_METHOD

// Copyright (c) 2024 Loupe (https://loupe.team), provided under the MIT License.
METHOD Connect
VAR_INPUT
END_VAR

// If Connection is already enabled, disable and disconnect
// Reference : https://infosys.beckhoff.com/content/1033/tf6760_tc3_iot_https_rest/9298409995.html?id=3568786990275794598
IF _connectionEnable THEN
	_connectionEnable := FALSE;
	_httpClient.Disconnect();
END_IF

_configureClient(configuration);
_connectionEnable := TRUE;

_methodConnectionStartCalled := TRUE;
END_METHOD

// Copyright (c) 2024 Loupe (https://loupe.team), provided under the MIT License.
METHOD Cyclic
VAR_INPUT
END_VAR

VAR
	retVal : BOOL;
	digestLocation : INT;
END_VAR

IF _connectionEnable THEN
	_httpClient.Execute();
	
	IF _httpClient.bError THEN
		errorID := _httpClient.hrErrorCode;
		errorMsg := 'Http Client object returned an error (see errorID)';
		_state := ABBLINKIN_STATE.ERROR;
	END_IF
END_IF

// Status
_sendingEnabled := _connectionEnable AND _httpClient.bConfigured AND NOT error;
readyForCmd := _sendingEnabled AND _authorized;


CASE _state OF 
	
	ABBLINKIN_STATE.IDLE:
		
		IF _sendingEnabled THEN
			IF _authorized THEN 
				
				// Check for existing request
				IF _currentRequest.pStatus <> 0	THEN 
					IF _currentRequest.pStatus^.busy THEN
						// Possible scenario: a request was sent, but a 401 Unauthorized was returned (causing re-auth steps). Here, we are retrying.	
						// Possible scenario: an error occured somewhere along the way	
						IF _numRequestAttempts < MAX_REQUESTS_ATTEMPTS THEN
							_state := ABBLINKIN_STATE.SEND_REQUEST;
						ELSE
							// Maximum number of requests sent -> terminate request
							_currentRequest.pStatus^.busy := FALSE;
							_currentRequest.pStatus^.done := FALSE;
							_currentRequest.pStatus^.error := TRUE;
							IF _currentRequest.pStatus^.errorMsg = '' THEN
								_currentRequest.pStatus^.errorMsg := 'Maximum number of request reached';
							END_IF
							MEMSET(ADR(_currentRequest), 0, SIZEOF(_currentRequest));	// Zero (i.e. terminate) current Request
						END_IF
					END_IF
				END_IF
				
				// Check if queue contains at least one request
				IF _state <> ABBLINKIN_STATE.SEND_REQUEST  AND NOT _requestQueue.empty THEN
					_currentRequest := _requestQueuePop();
					_numRequestAttempts := 0;
					_state := ABBLINKIN_STATE.SEND_REQUEST;
				END_IF
			ELSE
				// Start Auth sequence within state machine
				_state := ABBLINKIN_STATE.AUTH_SEND_REQUEST;
			END_IF
		END_IF
		
	ABBLINKIN_STATE.SEND_REQUEST:
		
		_setHeaders(ABBLINKIN_AUTH_HEADER_VALUE.NONE);
		retVal := _httpRequest.SendRequest(_currentRequest.uri, _httpClient, _currentRequest.httpMethod, ADR(_currentRequest.httpBody), INT_TO_UDINT(LEN(_currentRequest.httpBody)), _httpHeader);
		_numRequestAttempts := _numRequestAttempts + 1;
		
		IF retVal = FALSE THEN
			_currentRequest.pStatus^.busy := FALSE;
			_currentRequest.pStatus^.error := TRUE;
			_currentRequest.pStatus^.errorMsg := 'The request could not be sent';
			MEMSET(ADR(_currentRequest), 0, SIZEOF(_currentRequest));	// Zero (i.e. terminate) current Request
			
			_state := ABBLINKIN_STATE.IDLE;
		ELSE
			_state := ABBLINKIN_STATE.WAIT_FOR_RESONSE;
		END_IF
		
	ABBLINKIN_STATE.WAIT_FOR_RESONSE:
	
		IF _httpRequest.bError THEN
			_currentRequest.pStatus^.busy := FALSE;
			_currentRequest.pStatus^.error := TRUE;
			_currentRequest.pStatus^.errorID := _httpRequest.eErrorId;
			_currentRequest.pStatus^.errorMsg := CONCAT('Client request object error (see errorID) - ' , TO_STRING(_httpRequest.eErrorId));
			MEMSET(ADR(_currentRequest), 0, SIZEOF(_currentRequest));	// Zero (i.e. terminate) current Request
			
			_state := ABBLINKIN_STATE.IDLE;
		ELSIF _httpRequest.bBusy = FALSE THEN
			_state := ABBLINKIN_STATE.PROCESS_RESPONSE;
		END_IF
		
	ABBLINKIN_STATE.PROCESS_RESPONSE:
		
		CASE _httpRequest.nStatusCode OF 
		
			200..204 : // HTTP Success
			
				// Command-specific success-response-processing
				_callCommandSuccessHandler(_currentRequest, _httpRequest);
				
				// Write and close out current request status
				_currentRequest.pStatus^.busy := FALSE;
				_currentRequest.pStatus^.done := NOT _currentRequest.pStatus^.error; // Set done if error false
				MEMSET(ADR(_currentRequest), 0, SIZEOF(_currentRequest));	// Zero (i.e. terminate) current Request
				
				_state := ABBLINKIN_STATE.IDLE;
				
			401, 503: // HTTP Error - "Unauthorized" 
				
				// Go back to idle (will then proceed to auth steps before re-attempting)
				_authorized := FALSE;
				_state := ABBLINKIN_STATE.IDLE;
								
			400, 402..451:	// HTTP Client Error	
				_currentRequest.pStatus^.busy := FALSE;
				_currentRequest.pStatus^.error := TRUE;
				_currentRequest.pStatus^.errorID := _httpRequest.nStatusCode;
				_currentRequest.pStatus^.errorMsg := 'The Robot responded with an error (client error, 4xx). See errorID';
				MEMSET(ADR(_currentRequest), 0, SIZEOF(_currentRequest));	// Zero (i.e. terminate) current Request
				
				_state := ABBLINKIN_STATE.IDLE;
				
			500..502, 504..511: // HTTP Server Error
				_currentRequest.pStatus^.busy := FALSE;
				_currentRequest.pStatus^.error := TRUE;
				_currentRequest.pStatus^.errorID := _httpRequest.nStatusCode;
				_currentRequest.pStatus^.errorMsg := 'The Robot responded with an error (server error, 5xx). See errorID';
				MEMSET(ADR(_currentRequest), 0, SIZEOF(_currentRequest));	// Zero (i.e. terminate) current Request
				
				_state := ABBLINKIN_STATE.IDLE;
		END_CASE
	
	
	ABBLINKIN_STATE.AUTH_START:
		_auth.numAttempts := 0;
		_state := ABBLINKIN_STATE.AUTH_SEND_REQUEST;
		
	ABBLINKIN_STATE.AUTH_SEND_REQUEST:
		
		CASE configuration.rwsVersion OF
			ABBLINKIN_RWS_API_VERSION.V1:
				_setHeaders(ABBLINKIN_AUTH_HEADER_VALUE.NONE);
			ABBLINKIN_RWS_API_VERSION.V2:
				_setHeaders(ABBLINKIN_AUTH_HEADER_VALUE.BASIC);
		END_CASE
		
		retVal := _httpRequest.SendRequest(AUTH_URI, _httpClient, ETcIotHttpRequestType.HTTP_Get, 0, 0, _httpHeader);
		
		IF retVal = FALSE THEN
			errorID := 0;
			errorMsg := 'The Auth request could not be sent';
			_state := ABBLINKIN_STATE.ERROR;
		ELSE
			_state := ABBLINKIN_STATE.AUTH_WAIT_FOR_RESONSE;
		END_IF
		
	ABBLINKIN_STATE.AUTH_WAIT_FOR_RESONSE:
		
		IF _httpRequest.bError THEN
			errorID := _httpRequest.eErrorId;
			errorMsg := CONCAT('Client request object error (see errorID) - ' , TO_STRING(_httpRequest.eErrorId));
			_state := ABBLINKIN_STATE.ERROR;
		ELSIF _httpRequest.bBusy = FALSE THEN
			_state := ABBLINKIN_STATE.AUTH_PROCESS_RESPONSE;
		END_IF
		
	ABBLINKIN_STATE.AUTH_PROCESS_RESPONSE:
		
		_storeCookies(_httpRequest);
		
		CASE _httpRequest.nStatusCode OF 
		
			200..204 : // HTTP Success
				
				// Successfully authorized
				_authorized := TRUE;
				
				_state := ABBLINKIN_STATE.IDLE;
				
			401: // HTTP Error - "Unauthorized"
				
				CASE configuration.rwsVersion OF 
					ABBLINKIN_RWS_API_VERSION.V1:
						IF _httpRequest.GetHeaderField('WWW-Authenticate', ADR(_auth.wwwAuthContent), SIZEOF(_auth.wwwAuthContent)) THEN 
							_state := ABBLINKIN_STATE.AUTH_DIGEST_RESPONSE_CALCULATE;
						ELSE
							errorID := _httpRequest.nStatusCode;
							errorMsg := 'Unauthorized. No WWW-Authenticate header presented to digest.';
							_state := ABBLINKIN_STATE.ERROR;
						END_IF
					ABBLINKIN_RWS_API_VERSION.V2:
						errorID := _httpRequest.nStatusCode;
						errorMsg := 'Unauthorized. No WWW-Authenticate header presented to digest.';
						_state := ABBLINKIN_STATE.ERROR;
				END_CASE

				
			503:  
				// Note : You can get a 503 if you try to send the same credentials repeatedly instead of 
				// 		sending the http session cookies that the server provides after the first successful authentication			
				errorID := _httpRequest.nStatusCode;
				errorMsg := 'Authentication request recieved an error response (see errorID for HTTP code)';
				_state := ABBLINKIN_STATE.ERROR;
		ELSE			
			errorID := _httpRequest.nStatusCode;
			errorMsg := 'Authentication request recieved an error response (see errorID for HTTP code)';
			_state := ABBLINKIN_STATE.ERROR;			
		END_CASE
	
	ABBLINKIN_STATE.AUTH_DIGEST_RESPONSE_CALCULATE:
		// Calculate Digest parameters
		
		// Verify that DIGEST in header
		digestLocation := FIND(_auth.wwwAuthContent, 'Digest');
		IF digestLocation = 0 THEN
			errorID := 0;
			errorMsg := 'Digest not found in WWW-Authenticate header';
			_state := ABBLINKIN_STATE.ERROR;
		END_IF
		
		IF NOT error THEN
			// Extract parameter values from WWW-Authenticate header
			_auth.digest.realm	:= _parseWwwAuthForParameter('realm', _auth.wwwAuthContent);
			_auth.digest.qop	:= _parseWwwAuthForParameter('qop', _auth.wwwAuthContent);
			_auth.digest.nonce	:= _parseWwwAuthForParameter('nonce', _auth.wwwAuthContent);
			_auth.digest.opaque	:= _parseWwwAuthForParameter('opaque', _auth.wwwAuthContent);
		END_IF
		
		IF (_auth.digest.realm = '' OR
			_auth.digest.qop = '' OR
			_auth.digest.nonce = '' OR
			_auth.digest.opaque = '') THEN
			errorID := 0;
			errorMsg := 'Could not extract Digest parameters from WWW-Authenticate header';
			_state := ABBLINKIN_STATE.ERROR;
		END_IF
 
		IF NOT error THEN
			// Calculate Digest response
			_auth.digest.nc := '00000001';
			_auth.digest.cnonce := _generateCnonce();
			_auth.digest.response := _calculateDigestResponse(	username := configuration.rwsUsername,
																realm := _auth.digest.realm,
																password := configuration.rwsPassword,
																httpMethod := 'GET',
																uri := AUTH_URI,
																nonce := _auth.digest.nonce,
																nc := _auth.digest.nc,
																cnonce := _auth.digest.cnonce,
																qop := _auth.digest.qop);
			
			
			// Formulate request
			_auth.digest.authContent := 'Digest username="';
			concat2(ADR(_auth.digest.authContent), ADR(configuration.rwsUsername), ADR(_auth.digest.authContent), SIZEOF(_auth.digest.authContent));
			concat2(ADR(_auth.digest.authContent), ADR('", realm="'), ADR(_auth.digest.authContent), SIZEOF(_auth.digest.authContent));
			concat2(ADR(_auth.digest.authContent), ADR(_auth.digest.realm), ADR(_auth.digest.authContent), SIZEOF(_auth.digest.authContent));
			concat2(ADR(_auth.digest.authContent), ADR('", nonce="'), ADR(_auth.digest.authContent), SIZEOF(_auth.digest.authContent));
			concat2(ADR(_auth.digest.authContent), ADR(_auth.digest.nonce), ADR(_auth.digest.authContent), SIZEOF(_auth.digest.authContent));
			concat2(ADR(_auth.digest.authContent), ADR('", uri="'), ADR(_auth.digest.authContent), SIZEOF(_auth.digest.authContent));
			concat2(ADR(_auth.digest.authContent), ADR(AUTH_URI), ADR(_auth.digest.authContent), SIZEOF(_auth.digest.authContent));
			concat2(ADR(_auth.digest.authContent), ADR('", algorithm="MD5", qop="'), ADR(_auth.digest.authContent), SIZEOF(_auth.digest.authContent));
			concat2(ADR(_auth.digest.authContent), ADR(_auth.digest.qop), ADR(_auth.digest.authContent), SIZEOF(_auth.digest.authContent));
			concat2(ADR(_auth.digest.authContent), ADR('", nc="'), ADR(_auth.digest.authContent), SIZEOF(_auth.digest.authContent));
			concat2(ADR(_auth.digest.authContent), ADR(_auth.digest.nc), ADR(_auth.digest.authContent), SIZEOF(_auth.digest.authContent));
			concat2(ADR(_auth.digest.authContent), ADR('", cnonce="'), ADR(_auth.digest.authContent), SIZEOF(_auth.digest.authContent));
			concat2(ADR(_auth.digest.authContent), ADR(_auth.digest.cnonce), ADR(_auth.digest.authContent), SIZEOF(_auth.digest.authContent));
			concat2(ADR(_auth.digest.authContent), ADR('", response="'), ADR(_auth.digest.authContent), SIZEOF(_auth.digest.authContent));
			concat2(ADR(_auth.digest.authContent), ADR(_auth.digest.response), ADR(_auth.digest.authContent), SIZEOF(_auth.digest.authContent));
			concat2(ADR(_auth.digest.authContent), ADR('"'), ADR(_auth.digest.authContent), SIZEOF(_auth.digest.authContent));
			
			_state := ABBLINKIN_STATE.AUTH_DIGEST_RESPONSE_SEND;
		END_IF
	
	ABBLINKIN_STATE.AUTH_DIGEST_RESPONSE_SEND:
	
		_setHeaders(ABBLINKIN_AUTH_HEADER_VALUE.DIGEST);
		retVal := _httpRequest.SendRequest(AUTH_URI, _httpClient, ETcIotHttpRequestType.HTTP_Get, 0, 0, _httpHeader);
		
		IF retVal = FALSE THEN
			errorID := 0;
			errorMsg := 'The Auth Digest request could not be sent';
			_state := ABBLINKIN_STATE.ERROR;
		ELSE
			_state := ABBLINKIN_STATE.AUTH_WAIT_FOR_RESONSE;
		END_IF
		
	
	ABBLINKIN_STATE.ERROR:
		;// User must AckError, ConnectionStart, or ConnectionStop to reset out of Error state
	
END_CASE


// Handle Resetting Methods

IF _methodConnectionStartCalled THEN
	IF _httpClient.bError THEN
		errorID := _httpClient.hrErrorCode;
		errorMsg := 'Http Client object returned an error (see errorID)';
		_state := ABBLINKIN_STATE.ERROR;
	ELSE
		errorID := 0;
		errorMsg := '';
		_state := ABBLINKIN_STATE.IDLE;
	END_IF
	
	_methodConnectionStartCalled := FALSE;
END_IF

IF _methodConnectionStopCalled THEN
	errorID := 0;
	errorMsg := '';
	_state := ABBLINKIN_STATE.IDLE;
	
	_methodConnectionStopCalled := FALSE;
END_IF

IF _methodAckErrorCalled THEN
	errorID := 0;
	errorMsg := '';
	IF _state = ABBLINKIN_STATE.ERROR THEN
		_state := ABBLINKIN_STATE.IDLE;
	END_IF
	
	_methodAckErrorCalled := FALSE;
END_IF

// Set Error status
error := (_state = ABBLINKIN_STATE.ERROR);
END_METHOD

// Copyright (c) 2024 Loupe (https://loupe.team), provided under the MIT License.
METHOD Disconnect
VAR_INPUT
END_VAR

_httpClient.Disconnect();
_connectionEnable := FALSE;
_methodConnectionStopCalled := TRUE;
END_METHOD

// Copyright (c) 2024 Loupe (https://loupe.team), provided under the MIT License.
METHOD GetCtrlState : BOOL
VAR_INPUT
	pStatus : POINTER TO AbbLinkinRequestStatus_Typ;
	pResultState : POINTER TO STRING;
END_VAR

VAR
	request : AbbLinkinRequest_Typ;
END_VAR

VAR CONSTANT
	THIS_COMMAND_TYPE: ABBLINKIN_COMMAND_TYPE := ABBLINKIN_COMMAND_TYPE.GET_CTRL_STATE;
END_VAR

// Check for invalid status pointer
IF pStatus = 0 THEN
	GetCtrlState := FALSE;
	RETURN;
END_IF

// Clear Status
_clearRequestStatus(pStatus);

// Check for invalid results pointer
IF pResultState = 0 THEN
	pStatus^.error := TRUE;
	pStatus^.errorMsg := TO_STRING(THIS_COMMAND_TYPE);
	pStatus^.errorMsg := CONCAT(pStatus^.errorMsg, ' results pointer invalid.');
	GetCtrlState := FALSE;
	RETURN;
END_IF

request.pStatus := pStatus;
request.command := THIS_COMMAND_TYPE;
request.httpMethod :=  ETcIotHttpRequestType.HTTP_Get;

CASE configuration.rwsVersion OF
	ABBLINKIN_RWS_API_VERSION.V1:
		request.uri := '/rw/panel/ctrlstate?json=1';

	ABBLINKIN_RWS_API_VERSION.V2:	
		request.uri := '/rw/panel/ctrl-state';
END_CASE

request.results.pDataString := pResultState;

// Add Request to Queue, and Set Busy (or Error) Status
IF _requestQueueAdd(request) THEN
	pStatus^.busy := TRUE;
	GetCtrlState := TRUE;
ELSE
	pStatus^.error := TRUE;
	pStatus^.errorMsg := TO_STRING(THIS_COMMAND_TYPE);
	pStatus^.errorMsg := CONCAT(pStatus^.errorMsg, ' could not be added to request Queue');
	GetCtrlState := FALSE;
END_IF
END_METHOD

// Copyright (c) 2024 Loupe (https://loupe.team), provided under the MIT License.
METHOD GetIOAnalog : BOOL
VAR_INPUT
	signal : STRING;
	pStatus : POINTER TO AbbLinkinRequestStatus_Typ;
	pResult : POINTER TO LREAL;
END_VAR

GetIOAnalog := _getIO(signal, pStatus, pResultBOOL := 0, pResultDINT := 0, pResultLREAL := pResult);
END_METHOD

// Copyright (c) 2024 Loupe (https://loupe.team), provided under the MIT License.
METHOD GetIODigital : BOOL
VAR_INPUT
	signal : STRING;
	pStatus : POINTER TO AbbLinkinRequestStatus_Typ;
	pResult : POINTER TO BOOL;
END_VAR

GetIODigital := _getIO(signal, pStatus, pResultBOOL := pResult, pResultDINT := 0, pResultLREAL := 0);
END_METHOD

// Copyright (c) 2024 Loupe (https://loupe.team), provided under the MIT License.
METHOD GetIOGroup : BOOL
VAR_INPUT
	signal : STRING;
	pStatus : POINTER TO AbbLinkinRequestStatus_Typ;
	pResult : POINTER TO DINT;
END_VAR

GetIOGroup := _getIO(signal, pStatus, pResultBOOL := 0, pResultDINT := pResult, pResultLREAL := 0);
END_METHOD

// Copyright (c) 2024 Loupe (https://loupe.team), provided under the MIT License.
METHOD GetOpMode : BOOL
VAR_INPUT
	pStatus : POINTER TO AbbLinkinRequestStatus_Typ;
	pResultState : POINTER TO STRING;
END_VAR

VAR
	request : AbbLinkinRequest_Typ;
END_VAR

VAR CONSTANT
	THIS_COMMAND_TYPE: ABBLINKIN_COMMAND_TYPE := ABBLINKIN_COMMAND_TYPE.GET_OP_MODE;
END_VAR

// Check for invalid status pointer
IF pStatus = 0 THEN
	GetOpMode := FALSE;
	RETURN;
END_IF

// Clear Status
_clearRequestStatus(pStatus);

// Check for invalid results pointer
IF pResultState = 0 THEN
	pStatus^.error := TRUE;
	pStatus^.errorMsg := TO_STRING(THIS_COMMAND_TYPE);
	pStatus^.errorMsg := CONCAT(pStatus^.errorMsg, ' results pointer invalid.');
	GetOpMode := FALSE;
	RETURN;
END_IF

request.pStatus := pStatus;
request.command := THIS_COMMAND_TYPE;
request.httpMethod :=  ETcIotHttpRequestType.HTTP_Get;

CASE configuration.rwsVersion OF
	ABBLINKIN_RWS_API_VERSION.V1:
		request.uri := '/rw/panel/opmode?json=1';

	ABBLINKIN_RWS_API_VERSION.V2:	
		request.uri := '/rw/panel/opmode';
END_CASE

request.results.pDataString := pResultState;

// Add Request to Queue, and Set Busy (or Error) Status
IF _requestQueueAdd(request) THEN
	pStatus^.busy := TRUE;
	GetOpMode := TRUE;
ELSE
	pStatus^.error := TRUE;
	pStatus^.errorMsg := TO_STRING(THIS_COMMAND_TYPE);
	pStatus^.errorMsg := CONCAT(pStatus^.errorMsg, ' could not be added to request Queue');
	GetOpMode := FALSE;
END_IF
END_METHOD

// Copyright (c) 2024 Loupe (https://loupe.team), provided under the MIT License.
METHOD GetRapidState : BOOL
VAR_INPUT
	pStatus : POINTER TO AbbLinkinRequestStatus_Typ;
	pResultState : POINTER TO STRING;
END_VAR

VAR
	request : AbbLinkinRequest_Typ;
END_VAR

VAR CONSTANT
	THIS_COMMAND_TYPE: ABBLINKIN_COMMAND_TYPE := ABBLINKIN_COMMAND_TYPE.GET_RAPID_STATE;
END_VAR

// Check for invalid status pointer
IF pStatus = 0 THEN
	GetRapidState := FALSE;
	RETURN;
END_IF

// Clear Status
_clearRequestStatus(pStatus);

// Check for invalid results pointer
IF pResultState = 0 THEN
	pStatus^.error := TRUE;
	pStatus^.errorMsg := TO_STRING(THIS_COMMAND_TYPE);
	pStatus^.errorMsg := CONCAT(pStatus^.errorMsg, ' results pointer invalid.');
	GetRapidState := FALSE;
	RETURN;
END_IF

request.pStatus := pStatus;
request.command := THIS_COMMAND_TYPE;
request.httpMethod :=  ETcIotHttpRequestType.HTTP_Get;

CASE configuration.rwsVersion OF
	ABBLINKIN_RWS_API_VERSION.V1:
		request.uri := '/rw/rapid/execution?json=1';

	ABBLINKIN_RWS_API_VERSION.V2:	
		request.uri := '/rw/rapid/execution';
END_CASE

request.results.pDataString := pResultState;

// Add Request to Queue, and Set Busy (or Error) Status
IF _requestQueueAdd(request) THEN
	pStatus^.busy := TRUE;
	GetRapidState := TRUE;
ELSE
	pStatus^.error := TRUE;
	pStatus^.errorMsg := TO_STRING(THIS_COMMAND_TYPE);
	pStatus^.errorMsg := CONCAT(pStatus^.errorMsg, ' could not be added to request Queue');
	GetRapidState := FALSE;
END_IF
END_METHOD

// Copyright (c) 2024 Loupe (https://loupe.team), provided under the MIT License.
METHOD GetSymbolBool : BOOL
VAR_INPUT
	symbolUrl : STRING;
	pStatus : POINTER TO AbbLinkinRequestStatus_Typ;
	pResult : POINTER TO BOOL;
END_VAR

GetSymbolBool := _getSymbol(symbolUrl, pStatus, pResultBool := pResult, pResultLreal := 0, pResultString := 0);
END_METHOD

// Copyright (c) 2024 Loupe (https://loupe.team), provided under the MIT License.
METHOD GetSymbolNum : BOOL
VAR_INPUT
	symbolUrl : STRING;
	pStatus : POINTER TO AbbLinkinRequestStatus_Typ;
	pResult : POINTER TO LREAL;
END_VAR

GetSymbolNum := _getSymbol(symbolUrl, pStatus, pResultBool := 0, pResultLreal := pResult, pResultString := 0);
END_METHOD

// Copyright (c) 2024 Loupe (https://loupe.team), provided under the MIT License.
METHOD GetSymbolString : BOOL
VAR_INPUT
	symbolUrl : STRING;
	pStatus : POINTER TO AbbLinkinRequestStatus_Typ;
	pResult : POINTER TO STRING;
END_VAR

GetSymbolString := _getSymbol(symbolUrl, pStatus, pResultBool := 0, pResultLreal := 0, pResultString := pResult);
END_METHOD

// Copyright (c) 2024 Loupe (https://loupe.team), provided under the MIT License.
METHOD PowerOff : BOOL
VAR_INPUT
	pStatus : POINTER TO AbbLinkinRequestStatus_Typ;
END_VAR

VAR
	request : AbbLinkinRequest_Typ;
END_VAR

VAR CONSTANT
	THIS_COMMAND_TYPE: ABBLINKIN_COMMAND_TYPE := ABBLINKIN_COMMAND_TYPE.POWER_OFF;
END_VAR
IF pStatus = 0 THEN
	PowerOff := FALSE;
	RETURN;
END_IF

// Clear Status
_clearRequestStatus(pStatus);

request.pStatus := pStatus;
request.command := THIS_COMMAND_TYPE;
request.httpMethod :=  ETcIotHttpRequestType.HTTP_POST;

CASE configuration.rwsVersion OF
	ABBLINKIN_RWS_API_VERSION.V1:
		request.uri := '/rw/panel/ctrlstate?action=setctrlstate&json=1';
		request.httpBody := 'ctrl-state=motoroff';

	ABBLINKIN_RWS_API_VERSION.V2:	
		request.uri := '/rw/panel/ctrl-state';
		request.httpBody := 'ctrl-state=motoroff';
		
END_CASE

// Add Request to Queue, and Set Busy (or Error) Status
IF _requestQueueAdd(request) THEN
	pStatus^.busy := TRUE;
	PowerOff := TRUE;
ELSE
	pStatus^.error := TRUE;
	pStatus^.errorMsg := TO_STRING(THIS_COMMAND_TYPE);
	pStatus^.errorMsg := CONCAT(pStatus^.errorMsg, ' could not be added to request Queue');
	PowerOff := FALSE;
END_IF
END_METHOD

// Copyright (c) 2024 Loupe (https://loupe.team), provided under the MIT License.
METHOD PowerOn : BOOL
VAR_INPUT
	pStatus : POINTER TO AbbLinkinRequestStatus_Typ;
END_VAR

VAR
	request : AbbLinkinRequest_Typ;
END_VAR

VAR CONSTANT
	THIS_COMMAND_TYPE: ABBLINKIN_COMMAND_TYPE := ABBLINKIN_COMMAND_TYPE.POWER_ON;
END_VAR
IF pStatus = 0 THEN
	PowerOn := FALSE;
	RETURN;
END_IF

// Clear Status
_clearRequestStatus(pStatus);

request.pStatus := pStatus;
request.command := THIS_COMMAND_TYPE;
request.httpMethod :=  ETcIotHttpRequestType.HTTP_POST;

CASE configuration.rwsVersion OF
	ABBLINKIN_RWS_API_VERSION.V1:
		request.uri := '/rw/panel/ctrlstate?action=setctrlstate&json=1';
		request.httpBody := 'ctrl-state=motoron';

	ABBLINKIN_RWS_API_VERSION.V2:	
		request.uri := '/rw/panel/ctrl-state';
		request.httpBody := 'ctrl-state=motoron';
		
END_CASE

// Add Request to Queue, and Set Busy (or Error) Status
IF _requestQueueAdd(request) THEN
	pStatus^.busy := TRUE;
	PowerOn := TRUE;
ELSE
	pStatus^.error := TRUE;
	pStatus^.errorMsg := TO_STRING(THIS_COMMAND_TYPE);
	pStatus^.errorMsg := CONCAT(pStatus^.errorMsg, ' could not be added to request Queue');
	PowerOn := FALSE;
END_IF
END_METHOD

// Copyright (c) 2024 Loupe (https://loupe.team), provided under the MIT License.
METHOD RapidReset : BOOL
VAR_INPUT
	pStatus : POINTER TO AbbLinkinRequestStatus_Typ;
END_VAR

VAR
	request : AbbLinkinRequest_Typ;
END_VAR

VAR CONSTANT
	THIS_COMMAND_TYPE: ABBLINKIN_COMMAND_TYPE := ABBLINKIN_COMMAND_TYPE.RAPID_RESET;
END_VAR
IF pStatus = 0 THEN
	RapidReset := FALSE;
	RETURN;
END_IF

// Clear Status
_clearRequestStatus(pStatus);

request.pStatus := pStatus;
request.command := THIS_COMMAND_TYPE;
request.httpMethod :=  ETcIotHttpRequestType.HTTP_POST;

CASE configuration.rwsVersion OF
	ABBLINKIN_RWS_API_VERSION.V1:
		request.uri := '/rw/rapid/execution?action=resetpp&json=1';
		request.httpBody := '';

	ABBLINKIN_RWS_API_VERSION.V2:	
		request.uri := '/rw/rapid/execution/resetpp?mastership=implicit';
		request.httpBody := '';
		
END_CASE

// Add Request to Queue, and Set Busy (or Error) Status
IF _requestQueueAdd(request) THEN
	pStatus^.busy := TRUE;
	RapidReset := TRUE;
ELSE
	pStatus^.error := TRUE;
	pStatus^.errorMsg := TO_STRING(THIS_COMMAND_TYPE);
	pStatus^.errorMsg := CONCAT(pStatus^.errorMsg, ' could not be added to request Queue');
	RapidReset := FALSE;
END_IF
END_METHOD

// Copyright (c) 2024 Loupe (https://loupe.team), provided under the MIT License.
METHOD RapidStart : BOOL
VAR_INPUT
	pStatus : POINTER TO AbbLinkinRequestStatus_Typ;
END_VAR

VAR
	request : AbbLinkinRequest_Typ;
END_VAR

VAR CONSTANT
	THIS_COMMAND_TYPE: ABBLINKIN_COMMAND_TYPE := ABBLINKIN_COMMAND_TYPE.RAPID_START;
END_VAR
IF pStatus = 0 THEN
	RapidStart := FALSE;
	RETURN;
END_IF

// Clear Status
_clearRequestStatus(pStatus);

request.pStatus := pStatus;
request.command := THIS_COMMAND_TYPE;
request.httpMethod :=  ETcIotHttpRequestType.HTTP_POST;

CASE configuration.rwsVersion OF
	ABBLINKIN_RWS_API_VERSION.V1:
		request.uri := '/rw/rapid/execution?action=start&json=1';
		request.httpBody := '';
		request.httpBody := CONCAT(request.httpBody, 'regain=continue');
		request.httpBody := CONCAT(request.httpBody, '&execmode=continue');
		request.httpBody := CONCAT(request.httpBody, '&condition=none');
		request.httpBody := CONCAT(request.httpBody, '&cycle=once');
		request.httpBody := CONCAT(request.httpBody, '&stopatbp=disabled');
		request.httpBody := CONCAT(request.httpBody, '&alltaskbytsp=false');

	ABBLINKIN_RWS_API_VERSION.V2:	
		request.uri := '/rw/rapid/execution/start?mastership=implicit';
		request.httpBody := '';
		request.httpBody := CONCAT(request.httpBody, 'regain=continue');
		request.httpBody := CONCAT(request.httpBody, '&execmode=continue');
		request.httpBody := CONCAT(request.httpBody, '&condition=none');
		request.httpBody := CONCAT(request.httpBody, '&cycle=once');
		request.httpBody := CONCAT(request.httpBody, '&stopatbp=disabled');
		request.httpBody := CONCAT(request.httpBody, '&alltaskbytsp=false');
		
END_CASE

// Add Request to Queue, and Set Busy (or Error) Status
IF _requestQueueAdd(request) THEN
	pStatus^.busy := TRUE;
	RapidStart := TRUE;
ELSE
	pStatus^.error := TRUE;
	pStatus^.errorMsg := TO_STRING(THIS_COMMAND_TYPE);
	pStatus^.errorMsg := CONCAT(pStatus^.errorMsg, ' could not be added to request Queue');
	RapidStart := FALSE;
END_IF
END_METHOD

// Copyright (c) 2024 Loupe (https://loupe.team), provided under the MIT License.
METHOD RapidStop : BOOL
VAR_INPUT
	pStatus : POINTER TO AbbLinkinRequestStatus_Typ;
END_VAR

VAR
	request : AbbLinkinRequest_Typ;
END_VAR

VAR CONSTANT
	THIS_COMMAND_TYPE: ABBLINKIN_COMMAND_TYPE := ABBLINKIN_COMMAND_TYPE.RAPID_STOP;
END_VAR
IF pStatus = 0 THEN
	RapidStop := FALSE;
	RETURN;
END_IF

// Clear Status
_clearRequestStatus(pStatus);

request.pStatus := pStatus;
request.command := THIS_COMMAND_TYPE;
request.httpMethod :=  ETcIotHttpRequestType.HTTP_POST;

CASE configuration.rwsVersion OF
	ABBLINKIN_RWS_API_VERSION.V1:
		request.uri := '/rw/rapid/execution?action=stop&json=1';
		request.httpBody := '';

	ABBLINKIN_RWS_API_VERSION.V2:	
		request.uri := '/rw/rapid/execution/stop';
		request.httpBody := '';
		
END_CASE

// Add Request to Queue, and Set Busy (or Error) Status
IF _requestQueueAdd(request) THEN
	pStatus^.busy := TRUE;
	RapidStop := TRUE;
ELSE
	pStatus^.error := TRUE;
	pStatus^.errorMsg := TO_STRING(THIS_COMMAND_TYPE);
	pStatus^.errorMsg := CONCAT(pStatus^.errorMsg, ' could not be added to request Queue');
	RapidStop := FALSE;
END_IF
END_METHOD

// Copyright (c) 2024 Loupe (https://loupe.team), provided under the MIT License.
METHOD SetIO : BOOL
VAR_INPUT
	signal : STRING;
	value : ANY;
	pStatus : POINTER TO AbbLinkinRequestStatus_Typ;
END_VAR
VAR
	request : AbbLinkinRequest_Typ;
	pBool : POINTER TO BOOL;
	pSint : POINTER TO SINT;
	pUsint : POINTER TO USINT;
	pInt : POINTER TO INT;
	pUint : POINTER TO UINT;
	pDint : POINTER TO DINT;
	pUdint : POINTER TO UDINT;
	pReal : POINTER TO REAL;
	pLreal : POINTER TO LREAL;
END_VAR

VAR CONSTANT
	THIS_COMMAND_TYPE: ABBLINKIN_COMMAND_TYPE := ABBLINKIN_COMMAND_TYPE.SET_IO;
END_VAR

// Check for invalid status pointer
IF pStatus = 0 THEN
	SetIO := FALSE;
	RETURN;
END_IF

// Clear Status
_clearRequestStatus(pStatus);

request.pStatus := pStatus;
request.command := THIS_COMMAND_TYPE;
request.httpMethod :=  ETcIotHttpRequestType.HTTP_POST;

CASE configuration.rwsVersion OF
	ABBLINKIN_RWS_API_VERSION.V1:
		request.uri := '/rw/iosystem/signals/';
		request.uri := concat(request.uri, signal);
		request.uri := concat(request.uri, '?action=set');
		
	ABBLINKIN_RWS_API_VERSION.V2:
		request.uri := '/rw/iosystem/signals/';
		request.uri := concat(request.uri, signal);
		request.uri := concat(request.uri, '/set-value');

END_CASE

request.httpBody := 'lvalue=';
CASE value.TypeClass OF 
	__SYSTEM.TYPE_CLASS.TYPE_BOOL:
		pBool := value.pValue;
		IF pBool^ THEN
			request.httpBody := CONCAT(request.httpBody, '1');
		ELSE
			request.httpBody := CONCAT(request.httpBody, '0');
		END_IF
		
	__SYSTEM.TYPE_CLASS.TYPE_SINT:
		pSint := value.pValue;
		request.httpBody := CONCAT(request.httpBody, SINT_TO_STRING(pSint^));
	__SYSTEM.TYPE_CLASS.TYPE_USINT:
		pUsint := value.pValue;
		request.httpBody := CONCAT(request.httpBody, USINT_TO_STRING(pUsint^));
	__SYSTEM.TYPE_CLASS.TYPE_INT:
		pInt := value.pValue;
		request.httpBody := CONCAT(request.httpBody, INT_TO_STRING(pInt^));
	__SYSTEM.TYPE_CLASS.TYPE_UINT:
		pUint := value.pValue;
		request.httpBody := CONCAT(request.httpBody, UINT_TO_STRING(pUint^));
	__SYSTEM.TYPE_CLASS.TYPE_DINT:
		pDint := value.pValue;
		request.httpBody := CONCAT(request.httpBody, DINT_TO_STRING(pDint^));
	__SYSTEM.TYPE_CLASS.TYPE_UDINT:
		pUdint := value.pValue;
		request.httpBody := CONCAT(request.httpBody, UDINT_TO_STRING(pUdint^));
		
	__SYSTEM.TYPE_CLASS.TYPE_REAL:
		pReal := value.pValue;
		request.httpBody := CONCAT(request.httpBody, REAL_TO_STRING(pReal^));
	__SYSTEM.TYPE_CLASS.TYPE_LREAL:
		pLreal := value.pValue;
		request.httpBody := CONCAT(request.httpBody, LREAL_TO_STRING(pLreal^));
		
ELSE
	pStatus^.error := TRUE;
	pStatus^.errorMsg := TO_STRING(THIS_COMMAND_TYPE);
	pStatus^.errorMsg := CONCAT(pStatus^.errorMsg, ' was passed an unsupported "value" datatype');
	SetIO := FALSE;
	RETURN;
END_CASE

// Add Request to Queue, and Set Busy (or Error) Status
IF _requestQueueAdd(request) THEN
	pStatus^.busy := TRUE;
	SetIO := TRUE;
ELSE
	pStatus^.error := TRUE;
	pStatus^.errorMsg := TO_STRING(THIS_COMMAND_TYPE);
	pStatus^.errorMsg := CONCAT(pStatus^.errorMsg, ' could not be added to request Queue');
	SetIO := FALSE;
END_IF
END_METHOD

// Copyright (c) 2024 Loupe (https://loupe.team), provided under the MIT License.
METHOD SetSymbol : BOOL
VAR_INPUT
	symbolUrl : STRING;
	value : ANY;
	pStatus : POINTER TO AbbLinkinRequestStatus_Typ;
END_VAR

VAR
	request : AbbLinkinRequest_Typ;
	pBool : POINTER TO BOOL;
	pSint : POINTER TO SINT;
	pUsint : POINTER TO USINT;
	pInt : POINTER TO INT;
	pUint : POINTER TO UINT;
	pDint : POINTER TO DINT;
	pUdint : POINTER TO UDINT;
	pReal : POINTER TO REAL;
	pLreal : POINTER TO LREAL;
	pString : POINTER TO STRING;
	pWString : POINTER TO WSTRING;
END_VAR

VAR CONSTANT
	THIS_COMMAND_TYPE: ABBLINKIN_COMMAND_TYPE := ABBLINKIN_COMMAND_TYPE.SET_SYMBOL;
END_VAR

// Check for invalid status pointer
IF pStatus = 0 THEN
	SetSymbol := FALSE;
	RETURN;
END_IF

// Clear Status
_clearRequestStatus(pStatus);

request.pStatus := pStatus;
request.command := THIS_COMMAND_TYPE;
request.httpMethod :=  ETcIotHttpRequestType.HTTP_POST;

CASE configuration.rwsVersion OF
	ABBLINKIN_RWS_API_VERSION.V1:
		request.uri := '/rw/rapid/symbol/data/';
		request.uri := concat(request.uri, symbolUrl);
		request.uri := concat(request.uri, '?action=set');
		
	ABBLINKIN_RWS_API_VERSION.V2:
		request.uri := '/rw/rapid/symbol/';
		request.uri := concat(request.uri, symbolUrl);
		request.uri := concat(request.uri, '/data?mastership=implicit');
		
END_CASE

request.httpBody := 'value=';
CASE value.TypeClass OF 
	__SYSTEM.TYPE_CLASS.TYPE_BOOL:
		pBool := value.pValue;
		IF pBool^ THEN
			request.httpBody := CONCAT(request.httpBody, 'TRUE');
		ELSE
			request.httpBody := CONCAT(request.httpBody, 'FALSE');
		END_IF
		
	__SYSTEM.TYPE_CLASS.TYPE_SINT:
		pSint := value.pValue;
		request.httpBody := CONCAT(request.httpBody, SINT_TO_STRING(pSint^));
	__SYSTEM.TYPE_CLASS.TYPE_USINT:
		pUsint := value.pValue;
		request.httpBody := CONCAT(request.httpBody, USINT_TO_STRING(pUsint^));
	__SYSTEM.TYPE_CLASS.TYPE_INT:
		pInt := value.pValue;
		request.httpBody := CONCAT(request.httpBody, INT_TO_STRING(pInt^));
	__SYSTEM.TYPE_CLASS.TYPE_UINT:
		pUint := value.pValue;
		request.httpBody := CONCAT(request.httpBody, UINT_TO_STRING(pUint^));
	__SYSTEM.TYPE_CLASS.TYPE_DINT:
		pDint := value.pValue;
		request.httpBody := CONCAT(request.httpBody, DINT_TO_STRING(pDint^));
	__SYSTEM.TYPE_CLASS.TYPE_UDINT:
		pUdint := value.pValue;
		request.httpBody := CONCAT(request.httpBody, UDINT_TO_STRING(pUdint^));
		
	__SYSTEM.TYPE_CLASS.TYPE_REAL:
		pReal := value.pValue;
		request.httpBody := CONCAT(request.httpBody, REAL_TO_STRING(pReal^));
	__SYSTEM.TYPE_CLASS.TYPE_LREAL:
		pLreal := value.pValue;
		request.httpBody := CONCAT(request.httpBody, LREAL_TO_STRING(pLreal^));
		
	__SYSTEM.TYPE_CLASS.TYPE_STRING:
		request.httpBody := CONCAT(request.httpBody, '"');
		pString := value.pValue;
		request.httpBody := CONCAT(request.httpBody, pString^);
		request.httpBody := CONCAT(request.httpBody, '"');
	__SYSTEM.TYPE_CLASS.TYPE_WSTRING:
		request.httpBody := CONCAT(request.httpBody, '"');
		pWString := value.pValue;
		request.httpBody := CONCAT(request.httpBody, WSTRING_TO_STRING(pWString^));
		request.httpBody := CONCAT(request.httpBody, '"');
		
ELSE
	pStatus^.error := TRUE;
	pStatus^.errorMsg := TO_STRING(THIS_COMMAND_TYPE);
	pStatus^.errorMsg := CONCAT(pStatus^.errorMsg, ' was passed an unsupported "value" datatype');
	SetSymbol := FALSE;
	RETURN;
END_CASE

// Add Request to Queue, and Set Busy (or Error) Status
IF _requestQueueAdd(request) THEN
	pStatus^.busy := TRUE;
	SetSymbol := TRUE;
ELSE
	pStatus^.error := TRUE;
	pStatus^.errorMsg := TO_STRING(THIS_COMMAND_TYPE);
	pStatus^.errorMsg := CONCAT(pStatus^.errorMsg, ' could not be added to request Queue');
	SetSymbol := FALSE;
END_IF
END_METHOD

END_FUNCTION_BLOCK

// ---- POUs/Example.TcPOU
// Copyright (c) 2024 Loupe (https://loupe.team), provided under the MIT License.
PROGRAM Example
VAR
	myRobotLink : TcAbbLinkin;
	initConfiguration : BOOL := TRUE;
	initConnection : BOOL := TRUE;
	userCommand_GetState : BOOL := TRUE;
	getStateStatus : AbbLinkinRequestStatus_Typ;
	currentState : STRING;
	output : STRING;
END_VAR

// Initialize configuration
IF initConfiguration THEN
	myRobotLink.configuration.rwsIpAddress := '127.0.0.1';
	myRobotLink.configuration.rwsTcpPort := 80;
	myRobotLink.configuration.rwsVersion := ABBLINKIN_RWS_API_VERSION.V2;
	myRobotLink.configuration.rwsUsername := 'Default User';
	myRobotLink.configuration.rwsPassword := 'robotics';
	myRobotLink.configuration.tlsAllowRwsCertSelfSigned := TRUE;
	
	initConfiguration := FALSE;
END_IF

myRobotLink.Cyclic();

/////////////////////////
// Connect
IF initConnection THEN
	myRobotLink.ConnectionStart();
	initConnection := FALSE;
END_IF

/////////////////////////
// Get State

// Send command
IF myRobotLink.readyForCmd AND userCommand_GetState THEN
	myRobotLink.GetRapidState(pStatus := ADR(getStateStatus), pResultState := ADR(currentState));
	userCommand_GetState := FALSE;
END_IF

// Process Results
IF getStateStatus.done THEN
	output := CONCAT('Current state is ', currentState);
ELSIF getStateStatus.error THEN
	output := 'An Error occured.';
END_IF

END_PROGRAM
